(* IEC 61131-3 sources: volt/packages/volt-lsp-iec/test-corpus/pro2193/Library Manager/System_VisuInputs, 11 files *)

(* ---- VISU_INPUTS_GVL.gvl ---- *)
VAR_GLOBAL
	G_STVISUTOGGLEINPUTKEY : STRING(15) := 'Toggle_Input';
	G_VISUBUTTONINPUT : VisuFbButtonInput;
	G_PTMOUSEPOSITION : VisuStructPoint;
END_VAR

(* ---- VISU_INPUTS_VERSIONS.gvl ---- *)
VAR_GLOBAL
	_VISUINPUTS_VERSION_LARGEROREQUAL_3_3_1_0 : INT := 0;
	_VISUINPUTS_VERSION_LARGEROREQUAL_3_3_2_0 : INT := 0;
END_VAR

(* ---- VISUINPUT_CHECKUPDATEELEMENTSTATEPOSSIBLE_DEPENDINGONCURRENTINPUT.pou ---- *)
FUNCTION VISUINPUT_CHECKUPDATEELEMENTSTATEPOSSIBLE_DEPENDINGONCURRENTINPUT : BOOL
VAR_INPUT
	IVE : IVisualElement;
	PINPUT2 : POINTER TO VisuFbInputBase2;
	IELEMNR : DINT;
	PCURRENTCLIENTDATA : POINTER TO VisuStructClientData;
END_VAR
END_FUNCTION

(* ---- VISU_TAPINPUT.pou ---- *)
FUNCTION_BLOCK VISU_TAPINPUT
VAR_INPUT
	PVARIABLE : POINTER TO BOOL;
	BTAPFALSE : BOOL;
	BTAPONENTERIFCAPTURED : BOOL;
	DIBITOFFSET : DINT := -1;
END_VAR
VAR_OUTPUT
	BVALUE : BOOL;
END_VAR
VAR
	_IARMEDVALUECLIENTINDEX : DINT := -1;
	_OWNINGELEMENT : IVisualElement;
END_VAR
END_FUNCTION_BLOCK

METHOD FB_EXIT : BOOL
VAR_INPUT
	BINCOPYCODE : BOOL;
END_VAR
END_METHOD

METHOD INITIALIZE : BOOL
END_METHOD

METHOD ONDOWN : BOOL
VAR_INPUT
	PCLIENTDATA : POINTER TO VisuStructClientData;
	IVEOWNING : IVisualElement;
END_VAR
END_METHOD

METHOD ONENTER : BOOL
VAR_INPUT
	PCLIENTDATA : POINTER TO VisuStructClientData;
	IVEOWNING : IVisualElement;
END_VAR
END_METHOD

METHOD ONLEAVE : BOOL
VAR_INPUT
	PCLIENTDATA : POINTER TO VisuStructClientData;
	IVEOWNING : IVisualElement;
END_VAR
END_METHOD

METHOD ONUP : BOOL
VAR_INPUT
	PCLIENTDATA : POINTER TO VisuStructClientData;
END_VAR
END_METHOD

METHOD PROTARMCLICK : BOOL
VAR_INPUT
	PCLIENTDATA : POINTER TO VisuStructClientData;
	BARM : BOOL;
END_VAR
END_METHOD

METHOD PROTISARMED : BOOL
VAR_INPUT
	PCLIENTDATA : POINTER TO VisuStructClientData;
END_VAR
END_METHOD

METHOD PROTRESET : BOOL
END_METHOD

METHOD PROTSET : BOOL
END_METHOD

(* ---- VISU_TAPINPUTCONVERTED.pou ---- *)
FUNCTION_BLOCK VISU_TAPINPUTCONVERTED EXTENDS Visu_TapInput
VAR_INPUT
	PSTVARIABLE : POINTER TO STRING;
END_VAR
VAR
	_ONLVARREF : IVisuOnlineVariable;
	_BARM : BOOL;
END_VAR
END_FUNCTION_BLOCK

METHOD RESETVARIABLES
END_METHOD

METHOD PRVREGISTERVARIABLE
END_METHOD

METHOD PROTARMCLICK : BOOL
VAR_INPUT
	PCLIENTDATA : POINTER TO VisuStructClientData;
	BARM : BOOL;
END_VAR
END_METHOD

METHOD PROTISARMED : BOOL
VAR_INPUT
	PCLIENTDATA : POINTER TO VisuStructClientData;
END_VAR
END_METHOD

METHOD PROTRESET : BOOL
END_METHOD

METHOD PROTSET : BOOL
END_METHOD

(* ---- VISU_TOGGLEINPUT.pou ---- *)
FUNCTION_BLOCK VISU_TOGGLEINPUT
VAR_INPUT
	PVARIABLE : POINTER TO BOOL;
	BTOGGLEONCAPTUREDUP : BOOL;
	DIBITOFFSET : DINT := -1;
END_VAR
VAR_OUTPUT
	BVALUE : BOOL;
END_VAR
VAR
	_OWNINGELEMENT : IVisualElement;
	_IARMEDVALUE : DINT := -1;
	_PTOGGLEINPUTKEY : POINTER TO STRING := ADR(Visu_Inputs_Gvl.g_stVisuToggleInputKey);
	_PCLIENTDATA : POINTER TO VisuStructClientData;
END_VAR
END_FUNCTION_BLOCK

METHOD FB_EXIT : BOOL
VAR_INPUT
	BINCOPYCODE : BOOL;
END_VAR
END_METHOD

METHOD INITIALIZE : BOOL
VAR_INPUT
	OWNINGELEMENT : IVisualElement;
END_VAR
END_METHOD

METHOD ONDOWN : BOOL
VAR_INPUT
	PTMOUSE : VisuStructPoint;
END_VAR
END_METHOD

METHOD ONDOWN2 : BOOL
VAR_INPUT
	PTMOUSE : VisuStructPoint;
	IVEOWNING : IVisualElement;
END_VAR
END_METHOD

METHOD ONENTER : BOOL
END_METHOD

METHOD ONENTER2 : BOOL
VAR_INPUT
	IVEOWNING : IVisualElement;
END_VAR
END_METHOD

METHOD ONLEAVE : BOOL
END_METHOD

METHOD ONLEAVE2 : BOOL
VAR_INPUT
	IVEOWNING : IVisualElement;
END_VAR
END_METHOD

METHOD ONUP : BOOL
VAR_INPUT
	PTMOUSE : VisuStructPoint;
END_VAR
END_METHOD

METHOD ONUP2 : BOOL
VAR_INPUT
	PTMOUSE : VisuStructPoint;
	IVEOWNING : IVisualElement;
END_VAR
END_METHOD

METHOD PRVGETBUTTONSTATE : BOOL
VAR_INPUT
	IVEOWNING : IVisualElement;
END_VAR
END_METHOD

METHOD PRVSETBUTTONSTATE : BOOL
VAR_INPUT
	BDOWN : BOOL;
	IVEOWNING : IVisualElement;
END_VAR
END_METHOD

METHOD PROTGETARMED : BOOL
VAR_INPUT
	IVEOWNING : IVisualElement;
END_VAR
END_METHOD

METHOD PROTSETARMED : BOOL
VAR_INPUT
	BARM : BOOL;
	IVEOWNING : IVisualElement;
END_VAR
END_METHOD

METHOD PROTTOGGLE : BOOL
END_METHOD

(* ---- VISU_TOGGLEINPUTCONVERTED.pou ---- *)
FUNCTION_BLOCK VISU_TOGGLEINPUTCONVERTED EXTENDS Visu_ToggleInput
VAR_INPUT
	PSTVARIABLE : POINTER TO STRING;
END_VAR
VAR
	_ONLVARREF : IVisuOnlineVariable;
	_BARM : BOOL;
END_VAR
END_FUNCTION_BLOCK

METHOD RESETVARIABLES
END_METHOD

METHOD PRVREGISTERVARIABLE
END_METHOD

METHOD PROTGETARMED : BOOL
VAR_INPUT
	IVEOWNING : IVisualElement;
END_VAR
END_METHOD

METHOD PROTSETARMED : BOOL
VAR_INPUT
	BARM : BOOL;
	IVEOWNING : IVisualElement;
END_VAR
END_METHOD

METHOD PROTTOGGLE : BOOL
END_METHOD

(* ---- VISUFBBUTTONINPUT.pou ---- *)
FUNCTION_BLOCK VISUFBBUTTONINPUT EXTENDS VisuFbInputBase2
VAR
	M_TOGGLEINPUT : Visu_ToggleInput;
END_VAR
END_FUNCTION_BLOCK

METHOD EXECUTEMOUSEDOWN : BOOL
VAR_INPUT
	PCLIENTDATA : POINTER TO VisuStructClientData;
	PTMOUSE : VisuStructPoint;
	IVE : IVisualElement;
	DIELEMNR : DINT;
END_VAR
END_METHOD

METHOD EXECUTEMOUSEENTER : BOOL
VAR_INPUT
	PCLIENTDATA : POINTER TO VisuStructClientData;
	IVE : IVisualElement;
	DIELEMNR : DINT;
END_VAR
END_METHOD

METHOD EXECUTEMOUSELEAVE : BOOL
VAR_INPUT
	PCLIENTDATA : POINTER TO VisuStructClientData;
	IVE : IVisualElement;
	DIELEMNR : DINT;
END_VAR
END_METHOD

METHOD EXECUTEMOUSEUP : BOOL
VAR_INPUT
	PCLIENTDATA : POINTER TO VisuStructClientData;
	PTMOUSE : VisuStructPoint;
	IVE : IVisualElement;
	DIELEMNR : DINT;
END_VAR
END_METHOD

METHOD INITIALIZE : BOOL
VAR_INPUT
	PPARENTVISU : POINTER TO BYTE;
END_VAR
END_METHOD

METHOD PROTINPUTDISABLED : BOOL
VAR_INPUT
	IVE : IVisualElement;
	PEVENT : POINTER TO VisuStructEvent;
END_VAR
END_METHOD

(* ---- VISUFBINPUTBASE2.pou ---- *)
FUNCTION_BLOCK VISUFBINPUTBASE2
VAR
	M_PPARENTVISU : POINTER TO BYTE;
	BDUMMY : BOOL;
END_VAR
END_FUNCTION_BLOCK

METHOD EXECUTEEVENT : BOOL
VAR_INPUT
	PEVENT : POINTER TO VisuStructEvent;
	PCLIENTDATA : POINTER TO VisuStructClientData;
	IVE : IVisualElement;
	DIELEMNR : DINT;
END_VAR
END_METHOD

METHOD EXECUTELOOSECAPTURE : BOOL
VAR_INPUT
	PCLIENTDATA : POINTER TO VisuStructClientData;
	IVE : IVisualElement;
	DIELEMNR : DINT;
END_VAR
END_METHOD

METHOD GETELEMENTINFO : DWORD
VAR_INPUT
	PCLIENTDATA : POINTER TO VisuStructClientData;
	IVE : IVisualElement;
	DIELEMNR : DINT;
END_VAR
END_METHOD

METHOD HANDLEKEYEVENTIF : BOOL
VAR_INPUT
	PEVENT : POINTER TO VisuStructEvent;
	PCLIENTDATA : POINTER TO VisuStructClientData;
END_VAR
END_METHOD

METHOD INITIALIZE : BOOL
VAR_INPUT
	PPARENTVISU : POINTER TO BYTE;
END_VAR
END_METHOD

METHOD SETINPUTDELEGATE
VAR_INPUT
	INPUTDELEGATE : BOOL;
END_VAR
END_METHOD

METHOD ABSTRGETDEFAULTCURSOR : VisuEnumCursor
VAR_INPUT
	IVE : IVisualElement;
	DIELEMNR : DINT;
END_VAR
END_METHOD

METHOD PRVCHECKMOUSEOWNERSHIPEVENTS : BOOL
VAR_INPUT
	PEVENT : POINTER TO VisuStructEvent;
	PCLIENTDATA : POINTER TO VisuStructClientData;
	IVE : IVisualElement;
	DIELEMNR : DINT;
END_VAR
END_METHOD

METHOD PRVCONTAINSPOINT : BOOL
VAR_INPUT
	PT : VisuStructPoint;
	RSIMPLERECT : VisuStructSimpleRectangle;
	PCLIENTDATA : POINTER TO VisuStructClientData;
END_VAR
END_METHOD

METHOD PRVFORWARDEVENT : BOOL
VAR_INPUT
	PEVENT : POINTER TO VisuStructEvent;
	PCLIENT : POINTER TO VisuStructClientData;
	BCAPTURED : BOOL;
	IVE : IVisualElement;
	DIELEMNR : DINT;
END_VAR
END_METHOD

METHOD PRVISTOOLTIPONLYELEMENT : BOOL
VAR_INPUT
	PCLIENT : POINTER TO VisuStructClientData;
	IVE : IVisualElement;
	DIELEMNR : DINT;
END_VAR
END_METHOD

METHOD PRVSETCURSORIFNECESSARY : BOOL
VAR_INPUT
	PEVENT : POINTER TO VisuStructEvent;
	PCLIENTDATA : POINTER TO VisuStructClientData;
	IVE : IVisualElement;
	DIELEMNR : DINT;
END_VAR
END_METHOD

METHOD PRVSETINPUTINFO : BOOL
VAR_INPUT
	PCLIENT : POINTER TO VisuStructClientData;
	DIELEMNR : DINT;
END_VAR
END_METHOD

METHOD PROTINPUTDISABLED : BOOL
VAR_INPUT
	IVE : IVisualElement;
	PEVENT : POINTER TO VisuStructEvent;
END_VAR
END_METHOD

METHOD EXECUTEDIALOGCLOSED : BOOL
VAR_INPUT
	PCLIENTDATA : POINTER TO VisuStructClientData;
	DIALOG : IVisualisationDialog;
	IVE : IVisualElement;
	DIELEMNR : DINT;
END_VAR
END_METHOD

METHOD EXECUTEKEYDOWN : BOOL
VAR_INPUT
	PCLIENTDATA : POINTER TO VisuStructClientData;
	DWKEYCODE : DWORD;
	DWFLAGS : DWORD;
END_VAR
END_METHOD

METHOD EXECUTEKEYUP : BOOL
VAR_INPUT
	PCLIENTDATA : POINTER TO VisuStructClientData;
	DWKEYCODE : DWORD;
	DWFLAGS : DWORD;
END_VAR
END_METHOD

METHOD EXECUTEMOUSECLICK : BOOL
VAR_INPUT
	PCLIENTDATA : POINTER TO VisuStructClientData;
	PTMOUSE : VisuStructPoint;
	IVE : IVisualElement;
	DIELEMNR : DINT;
END_VAR
END_METHOD

METHOD EXECUTEMOUSEDBLCLICK : BOOL
VAR_INPUT
	PCLIENTDATA : POINTER TO VisuStructClientData;
	PTMOUSE : VisuStructPoint;
	IVE : IVisualElement;
	DIELEMNR : DINT;
END_VAR
END_METHOD

METHOD EXECUTEMOUSEDOWN : BOOL
VAR_INPUT
	PCLIENTDATA : POINTER TO VisuStructClientData;
	PTMOUSE : VisuStructPoint;
	IVE : IVisualElement;
	DIELEMNR : DINT;
END_VAR
END_METHOD

METHOD EXECUTEMOUSEENTER : BOOL
VAR_INPUT
	PCLIENTDATA : POINTER TO VisuStructClientData;
	IVE : IVisualElement;
	DIELEMNR : DINT;
END_VAR
END_METHOD

METHOD EXECUTEMOUSELEAVE : BOOL
VAR_INPUT
	PCLIENTDATA : POINTER TO VisuStructClientData;
	IVE : IVisualElement;
	DIELEMNR : DINT;
END_VAR
END_METHOD

METHOD EXECUTEMOUSEMOVE : BOOL
VAR_INPUT
	PCLIENTDATA : POINTER TO VisuStructClientData;
	PTMOUSE : VisuStructPoint;
	IVE : IVisualElement;
	DIELEMNR : DINT;
END_VAR
END_METHOD

METHOD EXECUTEMOUSEUP : BOOL
VAR_INPUT
	PCLIENTDATA : POINTER TO VisuStructClientData;
	PTMOUSE : VisuStructPoint;
	IVE : IVisualElement;
	DIELEMNR : DINT;
END_VAR
END_METHOD

METHOD EXECUTEVALUECHANGED : BOOL
VAR_INPUT
	PCLIENTDATA : POINTER TO VisuStructClientData;
	IVE : IVisualElement;
	DIELEMNR : DINT;
END_VAR
END_METHOD

(* ---- VISUFBRECTANGULARINPUTELEMENT.pou ---- *)
FUNCTION_BLOCK VISUFBRECTANGULARINPUTELEMENT EXTENDS VisuFbRectangularElement
VAR_INPUT
	M_PINPUTHANDLER : POINTER TO VisuFbInputBase2;
END_VAR
VAR
	M_BENABLED : BOOL;
END_VAR
END_FUNCTION_BLOCK

METHOD ISSELECTABLE : BOOL
END_METHOD

METHOD PAINTSELECTION : BOOL
VAR_INPUT
	PCURRENTSELECTIONDATA : POINTER TO Visu_StructSelectionData;
	SELECTIONCOLORS : VisuStructColors;
	SELECTIONLOOK : VisuStructElementLook;
	IFRAMEOFFSET : INT;
	IPOSITIONINDEX : INT;
	DWPAINTFLAGS : DWORD;
END_VAR
END_METHOD

METHOD SELECTELEMENT : DWORD
VAR_INPUT
	PCLIENTDATA : POINTER TO VisuStructClientData;
	PCURRENTSELECTIONDATA : POINTER TO Visu_StructSelectionData;
	PNEWSELECTIONDATA : POINTER TO Visu_StructSelectionData;
	DWSELECTIONTYPE : DWORD;
	DWGROUPTYPE : DWORD;
	PPOSITION : POINTER TO ARRAY [0..9] OF INT;
	IVISUALELEMENT : IVisualElement;
	IELEMINDEX : INT;
	IELEMID : INT;
	IPOSITIONINDEX : INT;
END_VAR
END_METHOD

METHOD ELEMENTINFO : INT
VAR_INPUT
	PDATA : POINTER TO Visu_StructElementInfo;
END_VAR
END_METHOD

METHOD HANDLEINPUT : BOOL
VAR_INPUT
	PEVENT : POINTER TO VisuStructEvent;
END_VAR
END_METHOD

(* ---- VISUFBRECTANGULARINPUTELEMENT2.pou ---- *)
FUNCTION_BLOCK VISUFBRECTANGULARINPUTELEMENT2 EXTENDS VisuFbRectangularElement2
VAR_INPUT
	M_PINPUTHANDLER : POINTER TO VisuFbInputBase2;
END_VAR
VAR
	M_BENABLED : BOOL;
END_VAR
END_FUNCTION_BLOCK

METHOD ISSELECTABLE : BOOL
END_METHOD

METHOD PAINTSELECTION : BOOL
VAR_INPUT
	PCURRENTSELECTIONDATA : POINTER TO Visu_StructSelectionData;
	SELECTIONCOLORS : VisuStructColors;
	SELECTIONLOOK : VisuStructElementLook;
	IFRAMEOFFSET : INT;
	IPOSITIONINDEX : INT;
	DWPAINTFLAGS : DWORD;
END_VAR
END_METHOD

METHOD SELECTELEMENT : DWORD
VAR_INPUT
	PCLIENTDATA : POINTER TO VisuStructClientData;
	PCURRENTSELECTIONDATA : POINTER TO Visu_StructSelectionData;
	PNEWSELECTIONDATA : POINTER TO Visu_StructSelectionData;
	DWSELECTIONTYPE : DWORD;
	DWGROUPTYPE : DWORD;
	PPOSITION : POINTER TO ARRAY [0..9] OF INT;
	IVISUALELEMENT : IVisualElement;
	IELEMINDEX : INT;
	IELEMID : INT;
	IPOSITIONINDEX : INT;
END_VAR
END_METHOD

METHOD ELEMENTINFO : INT
VAR_INPUT
	PDATA : POINTER TO Visu_StructElementInfo;
END_VAR
END_METHOD

METHOD HANDLEINPUT : BOOL
VAR_INPUT
	PEVENT : POINTER TO VisuStructEvent;
END_VAR
END_METHOD
